Fanuc KAREL source: port_AOUT.kl

PROGRAM TP
%NOLOCKGROUP
VAR
 x: INTEGER
BEGIN
 x = AOUT[3]
END TP
